VISUALIZATION Visualization  // 1024x768
END_VISUALIZATION

(* stored: Version 1.1.0.1
   Visu Visualization: Id {7c61372d-3361-46af-9943-f078fd14077c} *)
